{attribute 'qualified_only'}
{attribute 'strict'}
TYPE E_WriteStep :
(
	Stay,
	GripperOpen,
	ZAxixZeroPotision,
	XYAxixZeroPotision,
	PenGripp,
	Write,
	ZAxixZeroPotision2,
	XYAxixZeroPotision2,
	PenRelease,
	
	//McFb停止時用
	CommandAborted,
	Error,
	Reset
);
END_TYPE

(* stored: Version 1.1.0.1, ProductVersion 3.1.4026.12
   DUT E_WriteStep: Id {16e812ee-dab1-4da6-a6de-e6d899740546} *)
